INTERFACE IXyTable EXTENDS ZApplication.IUnit

END_INTERFACE

(* stored: Version 1.1.0.1
   Itf IXyTable: Id {5cc24f3e-61c5-482a-aad5-731feb80256f} *)
